TYPE E_DfiWriterState :
(
	IDLE := 0,
	CONNECT := 10,
	BUILD := 20,
	EXECUTE := 30,
	COMMIT := 40,
	ERROR := 90,
	DB_LOST := 99
) DINT;
END_TYPE

(* stored: Version 1.1.0.1
   DUT E_DfiWriterState: Id {0aec29fb-7fd4-4acc-8406-d222039da23c} *)
